FUNCTION_BLOCK FB_SQLMode_ExecuteCommandWithData
VAR_INPUT
	bExecute : BOOL ;
	hDBID : UINT ;
	sCommandSql : STRING(512) ;
END_VAR
VAR_OUTPUT
	bCommandOk : BOOL ;
	sError : STRING ;
    aReadStruct : ARRAY[1..10] OF ST_Database;	
END_VAR
VAR
    fbSqlDatabase : FB_SQLDatabaseEvt(sNetID := '', tTimeout := T#5S);
	fbSqlCommand : FB_SQLCommandEvt(sNetID := '', tTimeout := T#180S) ;
    tcMessage    : I_TcMessage;	
    fbSqlResult : FB_SQLResultEvt(sNetID:='', tTimeout    := T#5S); 	
	nState : INT ;
	fbPulse : R_TRIG ;

END_VAR

fbPulse(CLK:= bExecute, Q=> );

IF fbPulse.Q THEN
	nState := 1;		
END_IF

CASE nState OF
		
	0: ; //PARADO / IDLE / INTERRUMPIDO
		
	1: //LIMPA O BUFFER / CLEAN BUFFER / LIMPIA EL BUFFER
		fbSqlResult.Release();
		nState := 10;	 
		sError := '' ;	
	
	10: //ABRIR CONEXAO / OPEN CONECTION / CONEXION ABIERTA
	
		IF fbSqlDatabase.Connect(1) THEN
			IF fbSqlDatabase.bError THEN
				nState := 210; 
			ELSE
				nState := 20; 
			END_IF
		END_IF
	
	20: //CRIAR COMANDO / CREATE COMMAND / CREAR COMANDO
	
		IF fbSqlDatabase.CreateCmd(ADR(fbSqlCommand)) THEN
			IF fbSqlDatabase.bError THEN
				nState := 220; 			
			ELSE
				nState := 30; 
			END_IF
		END_IF	
		
	30: //EXECUTA COMANDO / EXCUTE COMMAND / EJECUTAR COMANDO
	
		IF fbSQLCommand.ExecuteDataReturn(ADR(sCommandSql), SIZEOF(sCommandSql), ADR(fbSqlResult)) THEN
			IF fbSQLCommand.bError THEN
				nState := 230; 				
			ELSE
				tcMessage := fbSQLCommand.ipTcResult;
				nState := 40; 
			END_IF
		END_IF
	
	40: //RECEBE OS DADOS / RECEIVE DATA / RECIBIR LOS DATOS
		IF fbSqlResult.Read(2, 3, ADR(aReadStruct), SIZEOF(aReadStruct), FALSE, TRUE) THEN
			IF fbSqlResult.bError THEN
				nState := 240; 
			ELSE
				nState := 50; 
			END_IF
		END_IF
	
	50: 
		fbSqlResult.Release();
			IF fbSqlResult.bError THEN
				nState := 250; 
			ELSE
				nState := 60; 
				sError := 'OK' ;				
			END_IF
	
		
	60:
		IF fbSqlDatabase.Disconnect() THEN
			IF fbSqlDatabase.bError THEN
				nState := 255;
			ELSE
				nState := 0;
			END_IF
		END_IF
		
	210 : 
		sError := 'Error Connect' ;
		nState := 60;		

	220 : 
		sError := 'Error Create Command' ;	
		nState := 60;	
		
	230: 
		sError := 'Error Execute Command' ;	
		nState := 60;	
		
	240: 
		sError := 'Error Read' ;			
		nState := 60;	
		
	250:
		sError := 'Error Release' ;		
		nState := 60;	
		
	260: 				
		sError := 'Error Disconect' ;	
		nState := 60;	
			
END_CASE

END_FUNCTION_BLOCK

(* stored: Version 1.1.0.1, ProductVersion 3.1.4024.12
   POU FB_SQLMode_ExecuteCommandWithData: Id {74584bf1-55a4-4104-81df-d17cf35ad8f7}, SpecialFunc None *)
